PROGRAM MAIN
VAR
END_VAR

Bases();
Lids();
Manipulator();
ControlPanel();

END_PROGRAM

(* stored: Version 1.1.0.1, ProductVersion 3.1.4024.9
   POU MAIN: Id {4675c6d2-396f-4c90-ba51-8852a4eba294}, SpecialFunc None *)
